ABB RobotStudio station: Proyecto_Final_B2_20210608-125324.rsstn

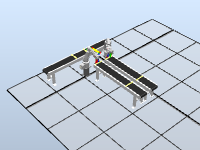
Station Station (saved by RobotStudio 20.4.9280.0)
Controller Controlador1, task T_ROB1: task frame (RAPID world) sits at (-70, -40, 300) mm, rotated rx 0 ry 0 rz -90 deg in the station
Controller Controlador1
  mechanical unit ROB_1: IRB120_3_58__Cuchara, 6 joints, base frame (0, 0, 0) mm
Controller Controlador2
  mechanical unit ROB_1: IRB120_3_58__Tenedor, 6 joints, base frame (-70, -860, 300) mm, rotated rx 0 ry 0 rz 90 deg
Layout (positions relative to the parent item):
  - Conveyor_Cuchara [part]
  - Conveyor_Tenedor [part]
  - Conveyor_Caja [part]
  - Cuchara [part] at (1956.71, -257.62, 505.45) mm, rotated rx 8.96 ry 0.3 rz 0.17 deg
  - Tenedor [part] at (1956.8, -630.69, 505.24) mm, rotated rx 0.08 ry 0.41 rz 0.06 deg
  - Logica_Conveyor_Cuchara [smart component]
      connections:
        LineSensor_Cuchara1.SensorOut -> Source_Cuchara.Execute
        LineSensor_Cuchara2.SensorOut -> PhysicsControl_Cuchara.SurfaceVelocityEnabled
    - LineSensor_Cuchara1 [smart component, from Components\LineSensor.rslib]
        properties: Start=[1.5 -0.39 0.508]; End=[1.5 -0.11 0.508]; Radius=0.003; SensedPart=(none); SensedPoint=[0 0 0]
      - _sensorPart_ [part]
    - Source_Cuchara [smart component, from Components\Source.rslib]
        properties: Source=Cuchara; Copy=(none); Parent=(none); Position=[1.957 -0.257623 0.505]; Orientation=[0 0 0]; Transient=true; PhysicsBehavior=3
    - LineSensor_Cuchara2 [smart component, from Components\LineSensor.rslib]
        properties: Start=[0.25 -0.39 0.508]; End=[0.25 -0.11 0.508]; Radius=0; SensedPart=(none); SensedPoint=[0 0 0]
      - _sensorPart_ [part]
    - PhysicsControl_Cuchara [smart component, from Components\PhysicsControl.rslib]
        properties: Object=Conveyor_Cuchara; Behavior=1; SurfaceVelocity=0.3
  - Logica_Conveyor_Tenedor [smart component]
      connections:
        LineSensor_Tenedor.SensorOut -> Source_Tenedor.Execute
        LineSensor_3.SensorOut -> PhysicsControl_Tenedor.SurfaceVelocityEnabled
    - LineSensor_Tenedor [smart component, from Components\LineSensor.rslib]
        properties: Start=[1.5 -0.8 0.508]; End=[1.5 -0.52 0.508]; Radius=0.003; SensedPart=(none); SensedPoint=[0 0 0]
      - _sensorPart_ [part]
    - Source_Tenedor [smart component, from Components\Source.rslib]
        properties: Source=Tenedor; Copy=(none); Parent=(none); Position=[1.957 -0.630695 0.505]; Orientation=[0 0 0]; Transient=true; PhysicsBehavior=3
    - LineSensor_3 [smart component, from Components\LineSensor.rslib]
        properties: Start=[0.25 -0.8 0.508]; End=[0.25 -0.52 0.508]; Radius=0; SensedPart=(none); SensedPoint=[0 0 0]
      - _sensorPart_ [part]
    - PhysicsControl_Tenedor [smart component, from Components\PhysicsControl.rslib]
        properties: Object=Conveyor_Tenedor; Behavior=1; SurfaceVelocity=0.3
  - Base_R_Tenedor [part] at (-70, -860, 0) mm
  - Base_R_Cuchara [part] at (-70, -40, 0) mm
  - Caja [part] at (-446, -1850, 506) mm
  - Logica_Conveyor_Caja [smart component]
      connections:
        LineSensor_Caja1.SensorOut -> Source_Caja.Execute
        LineSensor_Caja2.SensorOut -> PhysicsControl_Caja.SurfaceVelocityEnabled
    - LineSensor_Caja1 [smart component, from Components\LineSensor.rslib]
        properties: Start=[-0.59 -1 0.515]; End=[-0.31 -1 0.515]; Radius=0.005; SensedPart=(none); SensedPoint=[0 0 0]
      - _sensorPart_ [part]
    - Source_Caja [smart component, from Components\Source.rslib]
        properties: Source=Caja; Copy=(none); Parent=(none); Position=[-0.446 -1.89 0.506]; Orientation=[0 0 0]; Transient=true; PhysicsBehavior=3
    - LineSensor_Caja2 [smart component, from Components\LineSensor.rslib]
        properties: Start=[-0.59 -0.565 0.515]; End=[-0.31 -0.565 0.515]; Radius=0.005; SensedPart=(none); SensedPoint=[0 0 0]
      - _sensorPart_ [part]
    - PhysicsControl_Caja [smart component, from Components\PhysicsControl.rslib]
        properties: Object=Conveyor_Caja; Behavior=1; SurfaceVelocity=0.3
  - IRB120_3_58__Cuchara [mechanism, from Robots\IRB120_3_58_G_01.rslib] at (-70, -40, 300) mm, rotated rx 0 ry 0 rz -90 deg; joint values [1.015, 0.3085, 0.4252, 0, 0.837, 1.015] (rad or m)
  - IRB120_3_58__Tenedor [mechanism, from Robots\IRB120_3_58_G_01.rslib] at (-70, -860, 300) mm, rotated rx 0 ry 0 rz 90 deg; joint values [-1.0232, 0.2988, 0.4379, 0, 0.8341, -1.0232] (rad or m)
  - Mi_Ventosa [smart component, from Proyecto local\1217c23c-7d3e-48fb-b7d3-d1b2005a3c2bMi_Ventosa.rslib] at (230, -226.32, 625) mm, rotated rx 180 ry 0 rz 90 deg
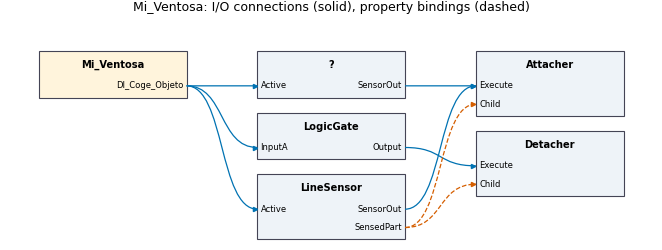
      connections:
        Mi_Ventosa.DI_Coge_Objeto -> ?.Active
        ?.SensorOut -> Attacher.Execute
        Mi_Ventosa.DI_Coge_Objeto -> LogicGate.InputA
        LogicGate.Output -> Detacher.Execute
        Mi_Ventosa.DI_Coge_Objeto -> LineSensor.Active
        LineSensor.SensorOut -> Attacher.Execute
        LineSensor.SensedPart => Attacher.Child
        LineSensor.SensedPart => Detacher.Child
    - Attacher [smart component, from Components\Attacher.rslib]
        properties: Parent=Ventosa; Flange=0; Child=(none); Mount=false; Offset=[0 0 0]; Orientation=[0 0 0]
    - Detacher [smart component, from Components\Detacher.rslib]
        properties: Child=(none); KeepPosition=true
    - Ventosa [mechanism, from Proyecto local\1217c23c-7d3e-48fb-b7d3-d1b2005a3c2bMi_Ventosa.rslib] at (0, 0, 0) mm
    - LogicGate [smart component, from Components\LogicGate.rslib]
        properties: Operator=NOT; Delay=0
    - LineSensor [smart component, from Components\LineSensor.rslib]
        properties: Start=[0 0 0.055]; End=[0 0 0.07]; Radius=0.001; SensedPart=(none); SensedPoint=[0 0 0]
      - _sensorPart_ [part]
    - Indicador [part, from Proyecto local\1217c23c-7d3e-48fb-b7d3-d1b2005a3c2bMi_Ventosa.rslib] at (-4.38, 0, 0) mm
  - Mi_Ventosa_2 [smart component, from Proyecto local\1217c23c-7d3e-48fb-b7d3-d1b2005a3c2bMi_Ventosa.rslib] at (229, -677.68, 625) mm, rotated rx 180 ry 0 rz -90 deg
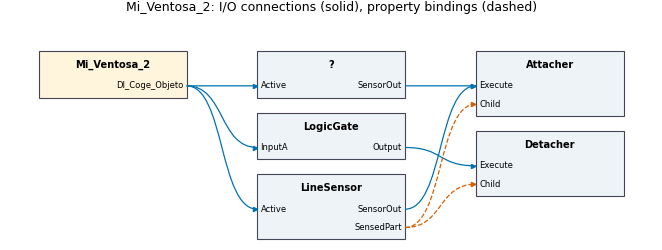
      connections:
        Mi_Ventosa_2.DI_Coge_Objeto -> ?.Active
        ?.SensorOut -> Attacher.Execute
        Mi_Ventosa_2.DI_Coge_Objeto -> LogicGate.InputA
        LogicGate.Output -> Detacher.Execute
        Mi_Ventosa_2.DI_Coge_Objeto -> LineSensor.Active
        LineSensor.SensorOut -> Attacher.Execute
        LineSensor.SensedPart => Attacher.Child
        LineSensor.SensedPart => Detacher.Child
    - Attacher [smart component, from Components\Attacher.rslib]
        properties: Parent=Ventosa; Flange=0; Child=(none); Mount=false; Offset=[0 0 0]; Orientation=[0 0 0]
    - Detacher [smart component, from Components\Detacher.rslib]
        properties: Child=(none); KeepPosition=true
    - Ventosa [mechanism, from Proyecto local\1217c23c-7d3e-48fb-b7d3-d1b2005a3c2bMi_Ventosa.rslib] at (0, 0, 0) mm
    - LogicGate [smart component, from Components\LogicGate.rslib]
        properties: Operator=NOT; Delay=0
    - LineSensor [smart component, from Components\LineSensor.rslib]
        properties: Start=[0 0 0.055]; End=[0 0 0.07]; Radius=0.001; SensedPart=(none); SensedPoint=[0 0 0]
      - _sensorPart_ [part]
    - Indicador [part, from Proyecto local\1217c23c-7d3e-48fb-b7d3-d1b2005a3c2bMi_Ventosa.rslib] at (-4.38, 0, 0) mm
  - Cuchara_2 [part] at (-162.14, -166.34, 4.12) mm, rotated rx 9.3 ry 0 rz -48.89 deg
  - Caja_2 [part] at (-446, -450, 506) mm
  - Tenedor_3 [part] at (153.79, -651.7, 2.94) mm, rotated rx 0 ry 0 rz 110.85 deg
Attachment: Mi_Ventosa is attached to IRB120_3_58__Cuchara / Link6
Attachment: Mi_Ventosa_2 is attached to IRB120_3_58__Tenedor / Link6
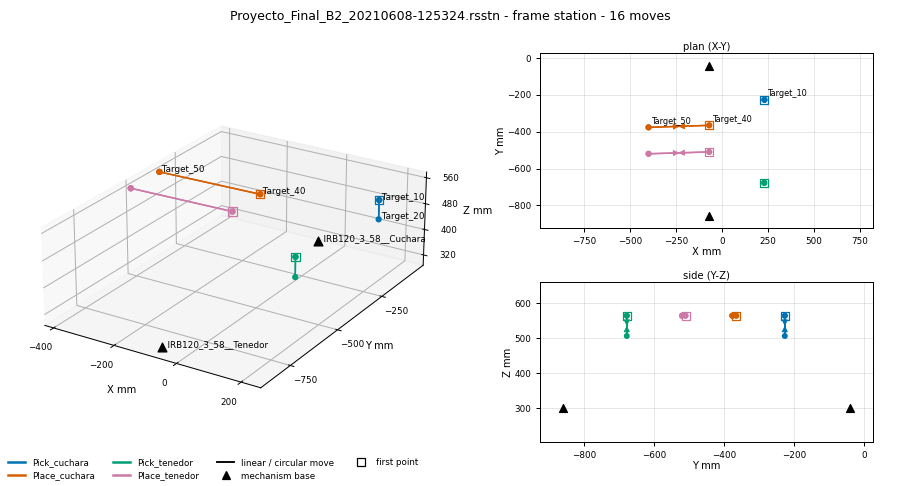
[picture p0: tool path of Proyecto_Final_B2_20210608-125324.rsstn in frame station, 16 of 16 moves have a stored position in this frame; points joined in program order, loops and branches not executed]
Targets, tools, work objects and paths stored in the station, written as RAPID:
! task T_ROB1
MODULE CalibData
  PERS tooldata TCP_Ventosa:=[TRUE,[[0,0,60],[1,0,0,0]],[0.1,[0,0,1],[1,0,0,0],0,0,0]];
  TASK PERS wobjdata Workobject_Cuchara:=[FALSE,TRUE,"",[[0,0,0],[1,0,0,0]],[[210,270,200],[1,0,0,0]]];
ENDMODULE

! task T_ROB1
MODULE Module1
  CONST robtarget Target_10:=[[-23.679886895,30.000008261,64.99887281],[0.000000136,-0.000000057,1,0.0000001],[0,-1,0,0],[9E+09,9E+09,9E+09,9E+09,9E+09,9E+09]];
  CONST robtarget Target_20:=[[-23.679890572,30.000002341,6.997147245],[-0.000000044,-0.000000082,1,-0.000000191],[0,-1,0,0],[9E+09,9E+09,9E+09,9E+09,9E+09,9E+09]];
  CONST robtarget Target_30:=[[-23.679995733,30.000024272,64.999939178],[0.000000004,0,1,0.000000007],[0,0,0,0],[9E+09,9E+09,9E+09,9E+09,9E+09,9E+09]];
  CONST robtarget Target_40:=[[115.150327174,-270.121311005,64.999168931],[-0.000000015,0.486157298,0.873871319,-0.000000026],[-1,-1,0,0],[9E+09,9E+09,9E+09,9E+09,9E+09,9E+09]];
  CONST robtarget Target_50:=[[126.149993321,-600.000025812,64.999544619],[0.000000008,0.4861829,0.873857075,-0.000000029],[-1,-1,0,0],[9E+09,9E+09,9E+09,9E+09,9E+09,9E+09]];
  CONST robtarget Target_51:=[[126.149993351,-600.000025877,64.999935931],[0,0.707106797,0.707106766,-0.000000016],[-1,-1,0,0],[9E+09,9E+09,9E+09,9E+09,9E+09,9E+09]];
  PROC Pick_cuchara()
    MoveJ Target_10,v600,z10,TCP_Ventosa\WObj:=Workobject_Cuchara;
    MoveL Target_20,v150,z1,TCP_Ventosa\WObj:=Workobject_Cuchara;
    MoveL Target_30,v150,z1,TCP_Ventosa\WObj:=Workobject_Cuchara;
  ENDPROC
  PROC Place_cuchara()
    MoveJ Target_40,v600,z10,TCP_Ventosa\WObj:=Workobject_Cuchara;
    MoveL Target_50,v300,z1,TCP_Ventosa\WObj:=Workobject_Cuchara;
    MoveL Target_51,v300,z1,TCP_Ventosa\WObj:=Workobject_Cuchara;
    MoveL Target_50,v300,z1,TCP_Ventosa\WObj:=Workobject_Cuchara;
    MoveL Target_40,v300,z1,TCP_Ventosa\WObj:=Workobject_Cuchara;
  ENDPROC
  PROC main()
    Pick_cuchara;
    Place_cuchara;
  ENDPROC
ENDMODULE

! task T_ROB1
MODULE CalibData
  PERS tooldata TCP_Ventosa:=[TRUE,[[0,0,60],[1,0,0,0]],[0.1,[0,0,1],[1,0,0,0],0,0,0]];
  TASK PERS wobjdata Workobject_Tenedor:=[FALSE,TRUE,"",[[200,-660,500],[0.707106781,0,0,-0.707106781]],[[0,0,0],[1,0,0,0]]];
ENDMODULE

! task T_ROB1
MODULE Module1
  CONST robtarget Target_10:=[[17.680001867,29.000010274,64.999168118],[0.000000019,1,-0.000000001,-0.000000013],[-1,0,-1,0],[9E+09,9E+09,9E+09,9E+09,9E+09,9E+09]];
  CONST robtarget Target_20:=[[17.680005,29.000006044,6.999955902],[0.000000007,1,0,-0.000000004],[-1,-1,-1,0],[9E+09,9E+09,9E+09,9E+09,9E+09,9E+09]];
  CONST robtarget Target_30:=[[17.680001867,29.000010274,64.999168118],[-0.000000019,1,-0.000000001,-0.000000013],[-1,0,-1,0],[9E+09,9E+09,9E+09,9E+09,9E+09,9E+09]];
  CONST robtarget Target_40:=[[-150.202171532,-270.144946432,64.99916005],[-0.000000007,0.871854368,0.489765211,0.000000003],[0,0,-1,0],[9E+09,9E+09,9E+09,9E+09,9E+09,9E+09]];
  CONST robtarget Target_50:=[[-140.200013899,-600.000004341,64.999949592],[0.000000013,0.871855673,0.489762887,0.000000004],[0,-1,-1,0],[9E+09,9E+09,9E+09,9E+09,9E+09,9E+09]];
  CONST robtarget Target_51:=[[-140.200013899,-600.000004341,64.999949592],[0.000000014,0.707106787,0.707106776,0],[0,-1,-1,0],[9E+09,9E+09,9E+09,9E+09,9E+09,9E+09]];
  PROC Pick_tenedor()
    MoveJ Target_10,v600,z10,TCP_Ventosa\WObj:=Workobject_Tenedor;
    MoveL Target_20,v150,z1,TCP_Ventosa\WObj:=Workobject_Tenedor;
    MoveL Target_30,v150,z1,TCP_Ventosa\WObj:=Workobject_Tenedor;
  ENDPROC
  PROC Place_tenedor()
    MoveJ Target_40,v600,z10,TCP_Ventosa\WObj:=Workobject_Tenedor;
    MoveL Target_50,v300,z1,TCP_Ventosa\WObj:=Workobject_Tenedor;
    MoveL Target_51,v300,z1,TCP_Ventosa\WObj:=Workobject_Tenedor;
    MoveL Target_50,v300,z1,TCP_Ventosa\WObj:=Workobject_Tenedor;
    MoveL Target_40,v300,z1,TCP_Ventosa\WObj:=Workobject_Tenedor;
  ENDPROC
  PROC main()
    Pick_tenedor;
    Place_tenedor;
  ENDPROC
ENDMODULE

